// TIA Portal V21 export
TYPE "Std_ForzaSendReceive"
   STRUCT
      Digitali : Array[0..31] of "Std_Segnale";
   END_STRUCT;
END_TYPE
